// TIA Portal V21 export
DATA_BLOCK "PHT Cycle"   // DB1201
{ S7_Optimized_Access := 'FALSE' }
// stored: AutoNumber false
   VAR
      Start : Bool;
      Stop : Bool;
      Abort : Bool;
      fault : Bool;
      Running : Bool;
      Selected : Bool;
      Actual_Min_Pressure : Real;
      Actual_Max_Pressure : Real;
      "Actual Stabilization Time" : DInt;
      "Actual Pressurise Hold Mins" : DInt;
      "Actual Pressurise Hold Secs" : DInt;
      "PHT Step Status int" : Int;
      "Step Status" : String[50];
      "Event Status" : String[50];
      print_event : Bool;
      "Startup Popup" : Bool;
      "Startup Popup Ack" : Bool;
      "Startup Popup Acked" : Bool;
      "Startup parameter popup" : Bool;
      "Abort Confirmation Popup" : Bool;
      "PHT Result" : Int;
      VesselSel : Int := 1;   // 1=Mv1, 2=Mv2, 3=Mv1&Mv2
      Result : String[50];
      Continue_Button : Bool;
      Abort_Button : Bool;
      "Actual Delay to Open Cai" : Int;
      PhtTemp : Bool;
      HOLD_FAIL : Bool;
      "Startup parameter popup No" : Bool;
      "Startup parameter popup Yes" : Bool;
      "Actual Delay to Open N2I" : Int;
      "N2IControl Valve" : Bool;
      EndOverPopup : Bool;
      EndOverPopupAck : Bool;
      CycleAbortEvent : Bool;
      "Abort confirmation popup Yes" : Bool;
      "Abort confirmation popup No" : Bool;
      InitialPressure : Real;
      FinalPressure : Real;
      HoldStartTimeLog : DTL;
      HoldEndTimeLog : DTL;
      TempTime : Time;
      RoundedTime : Time;
      TempMs : DInt;
      RoundedTime_Pos : Time;
      Hours : Int;
      Minutes : Int;
      Seconds : Int;
      TotalSecondsTag : DInt;
      PhtTimeDifference : Time;
   END_VAR
BEGIN
END_DATA_BLOCK
